	(* Init. NC parameter *)
		i:=1;
		(* Beckhoff *)
		IF sDeviceName = 'Beckhoff' THEN
			(*copy parameter value *)
			WHILE T_Axis.T_ParamFileObj[i].udiIdxGroup <> 0 DO
				CASE (T_Axis.T_ParamFileObj[i].udiIdxGroup - T_Axis.T_Config_Gen.udiNC_TaskIdxGrp) OF
				16#4000:	CASE T_Axis.T_ParamFileObj[i].udiIndexOffset OF
						(* Calibration velocity forward *)
						16#6:	T_Axis.T_Config_ObjFileValue.lrCalVelocityForward:=T_Axis.T_ParamFileObj[i].lrReal;
						(* Calibration velocity backward *)
						16#7:	T_Axis.T_Config_ObjFileValue.lrCalVelocityBackward:=T_Axis.T_ParamFileObj[i].lrReal;
						(* Maximum velocity *)
						16#27:	T_Axis.T_Config_ObjFileValue.lrMaxVelocity:=T_Axis.T_ParamFileObj[i].lrReal;
						(* Acceleration *)
						16#101:	T_Axis.T_Config_ObjFileValue.lrAcceleration:=T_Axis.T_ParamFileObj[i].lrReal;
						(* Decceleration *)
						16#102:	T_Axis.T_Config_ObjFileValue.lrDecceleration:=T_Axis.T_ParamFileObj[i].lrReal;
						(* Jerk *)
						16#103:	T_Axis.T_Config_ObjFileValue.lrJerk:=T_Axis.T_ParamFileObj[i].lrReal;
						END_CASE
				16#5000:	CASE T_Axis.T_ParamFileObj[i].udiIndexOffset OF
						(* Encoder scaling factor *)
						16#6:	T_Axis.T_Config_ObjFileValue.lrScaleFactor:=T_Axis.T_ParamFileObj[i].lrReal;
						(* SW limit negativ On/Off *)
						16#B:	T_Axis.T_Config_ObjFileValue.xSWLimitNeg:=REAL_TO_BOOL(T_Axis.T_ParamFileObj[i].lrReal);
						(* SW limit positiv On/Off *)
						16#C:	T_Axis.T_Config_ObjFileValue.xSWLimitPos:=REAL_TO_BOOL(T_Axis.T_ParamFileObj[i].lrReal);
						(* SW limit negativ value *)
						16#D:	T_Axis.T_Config_ObjFileValue.lrSWLimitNeg:=T_Axis.T_ParamFileObj[i].lrReal;
						(* SW limit position value *)
						16#E:	T_Axis.T_Config_ObjFileValue.lrSWLimitPos:=T_Axis.T_ParamFileObj[i].lrReal;
						END_CASE
				16#6000:;
				16#7000:;
				END_CASE
				(* next parameter *)
				i:=i+1;
			END_WHILE
		END_IF

		(* Maxon *)
		IF sDeviceName = 'Maxon' THEN
			(*copy parameter value *)
			WHILE T_Axis.T_ParamFileObj[i].udiIdxGroup <> 0 DO
				CASE T_Axis.T_ParamFileObj[i].udiIdxGroup  OF
				16#6083:	CASE T_Axis.T_ParamFileObj[i].udiIndexOffset OF
						(* Acceleration *)
						16#0:	T_Axis.T_Config_ObjFileValue.lrAcceleration:=T_Axis.T_ParamFileObj[i].lrReal;
						END_CASE
				16#6084:	CASE T_Axis.T_ParamFileObj[i].udiIndexOffset OF
						(* Decceleration *)
						16#0:	T_Axis.T_Config_ObjFileValue.lrDecceleration:=T_Axis.T_ParamFileObj[i].lrReal;
						END_CASE
				END_CASE
				(* next parameter *)
				i:=i+1;
			END_WHILE
		END_IF
		(* set flag done *)
		xBusy:=FALSE;
		xDone:=TRUE;
	END_IF;
END_FUNCTION_BLOCK

(* POU FB_HARDWARE/FBHW_AXIS_LIVEVALUES_BECKHOFF, ST *)
FUNCTION_BLOCK FBHW_AXIS_LIVEVALUES_BECKHOFF
VAR_INPUT
	uiActualTorque: UINT;
	arxDigitalInput: ARRAY[1..8] OF BOOL;
END_VAR
VAR_OUTPUT
END_VAR
VAR_IN_OUT
	T_Axis:ST_AXIS;
	T_AxisRefIn:NCTOPLC_AXLESTRUCT;
END_VAR
VAR
	i:INT;
END_VAR
(****************************************************************************************************************************************************)
(***********                                    This Functionblock read the actual value from the Beckhoff drive                                               ************)
(****************************************************************************************************************************************************)
(* return actual axis state *)
T_Axis.T_LiveValue.dwState:=T_AxisRefIn.nStateDWord;
(* return actual torque value *)
T_Axis.T_LiveValue.uiActualTorque:=uiActualTorque;
IF T_Axis.T_LiveValue.uiActualTorque > 16#7FFF THEN
	(* negativ value *)
	T_Axis.T_LiveValue.diActualTorqueCalc:=UINT_TO_DINT(T_Axis.T_LiveValue.uiActualTorque) - 65535;
ELSE
	(* positiv value *)
	T_Axis.T_LiveValue.diActualTorqueCalc:=UINT_TO_DINT(T_Axis.T_LiveValue.uiActualTorque);
END_IF
(* return actual velocity *)
T_Axis.T_LiveValue.lrActualVelocity:=T_AxisRefIn.fVeloIst;
(* ??? modif 06092005 *)
(* return actual position *)
IF T_Axis.T_Config_Gen.iTyp <>1 THEN
(* modulo position for rotativ axis*)
	T_Axis.T_LiveValue.lrActualPosition:=T_AxisRefIn.fModuloPosIst;
	T_Axis.T_LiveValue.lrActualPositionNotModulo:=T_AxisRefIn.fPosIst;
ELSE
(* counter value *)
	T_Axis.T_LiveValue.lrActualPosition:=T_AxisRefIn.fPosIst;
END_IF
T_Axis.T_LiveValue.lrSollPosition:=T_AxisRefIn.fPosSoll;
(* return actual position *)
(*T_Axis.T_LiveValue.lrActualPosition:=T_AxisRefIn.fPosIst;*)
(* ??? modif 06092005 *)
(* return the actual digital input state *)
T_Axis.T_LiveValue.bDigitalInput:=0;
FOR i := 0 TO 7 DO
	IF arxDigitalInput[i+1] THEN
		T_Axis.T_LiveValue.bDigitalInput:=T_Axis.T_LiveValue.bDigitalInput + MUX(i,1,2,4,8,16,32,64,128);
	END_IF
END_FOR;
END_FUNCTION_BLOCK

(* POU FB_HARDWARE/FBHW_AXIS_MULTI_BECKHOFF, ST *)
FUNCTION_BLOCK FBHW_AXIS_MULTI_BECKHOFF
VAR_INPUT
END_VAR
VAR_OUTPUT
END_VAR
VAR_IN_OUT
	T_AxisMaster:ST_AXIS;
	T_AxisSlave:ST_AXIS;
	T_AxisMasterRefIn:NCTOPLC_AXLESTRUCT;
	T_AxisSlaveRefIn:NCTOPLC_AXLESTRUCT;
END_VAR
VAR
(* block function *)
	fbAxisMasterSlaveOn:MC_GearIn;
	fbAxisMasterSlaveOff:MC_GearOut;
(* variable *)
	xGearIn:BOOL:=FALSE;
	xGearOut:BOOL:=FALSE;
	xConfirmResetFB:BOOL:=FALSE;
(* trigger *)
	RisingEdgeResetFB:R_TRIG;
	RisingEdgeExecute:R_TRIG;
END_VAR
(****************************************************************************************************************************************************)
(***********                                   This Functionblock is the driver for the Beckhoff Axis for Master/Slave                                      ************)
(****************************************************************************************************************************************************)
(* Reset block function *)
	RisingEdgeResetFB(CLK:=T_AxisMaster.T_CtrleMulti.xReset);
	IF RisingEdgeResetFB.Q THEN
	(* Init. block function *)
		fbAxisMasterSlaveOn(	Execute:=FALSE,
							Master:=T_AxisMasterRefIn,
							Slave:=T_AxisSlaveRefIn);
		fbAxisMasterSlaveOff(	Execute:=FALSE,
							Slave:=T_AxisSlaveRefIn);
	(* Init. variable *)
		xGearIn:=FALSE;
		xGearOut:=FALSE;
	(* init. structure *)
		T_AxisMaster.T_CtrleMulti.iFunction:=0;
		T_AxisMaster.T_CtrleMulti.iNumerator:=1;
		T_AxisMaster.T_CtrleMulti.uiDenominator:=1;
		T_AxisMaster.T_CtrleMulti.xDone:=FALSE;
		T_AxisMaster.T_CtrleMulti.xErr:=FALSE;
		T_AxisMaster.T_CtrleMulti.udiErrorID:=0;
		(* set done flag *)
		xConfirmResetFB:=TRUE;
		(* exit function bloc *)
		RETURN;
	ELSE
		IF xConfirmResetFB THEN
		(* confirm reset FB *)
			T_AxisMaster.T_CtrleMulti.xDone:=TRUE;
			T_AxisMaster.T_CtrleMulti.xErr:=FALSE;
			T_AxisMaster.T_CtrleMulti.udiErrorID:=0;
			(* reset variable *)
			xConfirmResetFB:=FALSE;
		END_IF
	END_IF

(* Execute *)
	RisingEdgeExecute(CLK:=T_AxisMaster.T_CtrleMulti.xExecute);
	IF RisingEdgeExecute.Q THEN
		CASE T_AxisMaster.T_CtrleMulti.iFunction OF
		(* activ master-slave *)
		1:	xGearIn:=TRUE;
		(* desactiv master-slave *)
		2: 	xGearOut:=TRUE;
		ELSE
		(* function not implemented *)
			T_AxisMaster.T_CtrleMulti.xDone:=FALSE;
			T_AxisMaster.T_CtrleMulti.xErr:=TRUE;
			T_AxisMaster.T_CtrleMulti.udiErrorID:=16#F000;
			(* exit FB *)
			RETURN;
		END_CASE
		(* Init. variable *)
		T_AxisMaster.T_CtrleMulti.xDone:=FALSE;
		T_AxisMaster.T_CtrleMulti.xErr:=FALSE;
		T_AxisMaster.T_CtrleMulti.udiErrorID:=0;
	END_IF

(* GearIn *)
	IF xGearIn THEN
		fbAxisMasterSlaveOn(	Execute:=TRUE,
							RatioNumerator:=T_AxisMaster.T_CtrleMulti.iNumerator,
							RatioDenominator:=T_AxisMaster.T_CtrleMulti.uiDenominator,
							Acceleration:=T_AxisMaster.T_CtrleSingle.lrAcceleration,
							Deceleration:=T_AxisMaster.T_CtrleSingle.lrDecceleration,
							Jerk:=T_AxisMaster.T_CtrleSingle.lrJerk,
							Master:=T_AxisMasterRefIn,
							Slave:=T_AxisSlaveRefIn);
		IF fbAxisMasterSlaveOn.InGear OR fbAxisMasterSlaveOn.Error THEN
			T_AxisMaster.T_CtrleMulti.xDone:= fbAxisMasterSlaveOn.InGear;
			T_AxisMaster.T_CtrleMulti.xErr:=fbAxisMasterSlaveOn.Error;
			T_AxisMaster.T_CtrleMulti.udiErrorID:=fbAxisMasterSlaveOn.ErrorID;
			(* set flag gearin off *)
			xGearIn:=FALSE;
		END_IF
	ELSE
		fbAxisMasterSlaveOn(	Execute:=FALSE,
							Master:=T_AxisMasterRefIn,
							Slave:=T_AxisSlaveRefIn);
	END_IF

(* GearOut *)
	IF xGearOut THEN
		fbAxisMasterSlaveOff(	Execute:=TRUE,
							Slave:=T_AxisSlaveRefIn);
		IF fbAxisMasterSlaveOff.Done OR fbAxisMasterSlaveOff.Error THEN
			T_AxisMaster.T_CtrleMulti.xDone:= fbAxisMasterSlaveOff.Done;
			T_AxisMaster.T_CtrleMulti.xErr:=fbAxisMasterSlaveOff.Error;
			T_AxisMaster.T_CtrleMulti.udiErrorID:=fbAxisMasterSlaveOff.ErrorID;
			(* set flag gearout off *)
			xGearOut:=FALSE;
		END_IF
	ELSE
		fbAxisMasterSlaveOff(	Execute:=FALSE,
							Slave:=T_AxisSlaveRefIn);
	END_IF
END_FUNCTION_BLOCK

(* POU FB_HARDWARE/FBHW_CYL_ANALOGCYLINDER, ST *)
FUNCTION_BLOCK FBHW_CYL_ANALOGCYLINDER
VAR_INPUT
	xCtrlePosOn:BOOL;
	xCtrlePosOff:BOOL;
	iAnalogIn:INT;
END_VAR
VAR_OUTPUT
	xCylinder:BOOL;
	iAnalogOut:INT;
END_VAR
VAR_IN_OUT
	T_Cylinder:ST_CYLINDER;
END_VAR
VAR
(* variable *)
	xConfirmResetFB: BOOL;
	xActivCtrle:BOOL;
	iStep:INT;
(* timer *)
	TimerOn:TON;
	TimerOff:TON;
	TimerPreOn:TON;
	TimerPreOff:TON;
	TimerOut:TON;
	TimerActiv: TON;
(* trigger *)
	RisingEdgeExecute:R_TRIG;
	RisingEdgeReset:R_TRIG;
	RisingEdgeActiv:R_TRIG;
	FallingEdgeActiv:F_TRIG;
	xFct3Activ: BOOL;
	xTmpFct3Activ: BOOL;
END_VAR
(****************************************************************************************************************************************************)
(***********                                       This Functionblock is the driver for the ToolTension Cylinder                                                    ************)
(****************************************************************************************************************************************************)
(* if function bloc set activ then Analog state will be transfered *)
	RisingEdgeActiv(CLK:=T_Cylinder.T_CtrleCyl.xFBActiv);
	FallingEdgeActiv(CLK:=T_Cylinder.T_CtrleCyl.xFBActiv);
	IF RisingEdgeActiv.Q OR FallingEdgeActiv.Q THEN
		iAnalogOut:=0;
		xCylinder:=NOT(T_Cylinder.T_Config.xActivState);
		T_Cylinder.T_CtrleCyl.T_AnalogCylinder.xActiv:= FALSE;
	END_IF
	(* transfer sensor state only if fb is activ *)
	IF T_Cylinder.T_CtrleCyl.xFBActiv THEN
		T_Cylinder.T_CtrleCyl.xStatePosOn:=xCtrlePosOn;
		T_Cylinder.T_CtrleCyl.xStatePosOff:=xCtrlePosOff;
	(* copy state value *)
		T_Cylinder.T_CtrleCyl.T_AnalogCylinder.iAnalogOut:=iAnalogOut;
	ELSE
	(* exit fb *)
		RETURN;
	END_IF

(* wait for reseting *)
	RisingEdgeReset(CLK:=T_Cylinder.T_CtrleCyl.xReset);
	IF RisingEdgeReset.Q THEN
		(* Init. timer *)
		TimerOn(IN:=TRUE,PT:=T#1ms);
		TimerOff(IN:=TRUE,PT:=T#1ms);
		TimerOut(IN:=TRUE,PT:=T#1ms);
		TimerPreOn(IN:=TRUE,PT:=T#1ms);
		TimerPreOff(IN:=TRUE,PT:=T#1ms);
		TimerActiv(IN:=TRUE,PT:=T#1ms);
	(* Init. variable *)
		xActivCtrle:=FALSE;
		iStep:=0;
		xFct3Activ:=FALSE;
		xTmpFct3Activ:=FALSE;
		T_Cylinder.T_CtrleCyl.T_AnalogCylinder.tDelayActiv:=T#0s;
		T_Cylinder.T_Config.tDelayPreOn:=T#0s;
		T_Cylinder.T_Config.tDelayPreOff:=T#0s;
	(* Init. structure *)
		T_Cylinder.T_CtrleCyl.iFunction:=0;
		T_Cylinder.T_CtrleCyl.T_AnalogCylinder.xActiv:= FALSE;
		xCylinder:=NOT(T_Cylinder.T_Config.xActivState);
		iAnalogOut:=0;
		T_Cylinder.T_CtrleCyl.xDone:=FALSE;
		T_Cylinder.T_CtrleCyl.xErr:=FALSE;
		T_Cylinder.T_CtrleCyl.udiErrorID:=16#0;
	(* confirm reset *)
		xConfirmResetFB:=TRUE;
	(* exit function *)
		RETURN;
	ELSE
		IF xConfirmResetFB THEN
		(* confirm reset FB *)
			T_Cylinder.T_CtrleCyl.xDone:=TRUE;
			T_Cylinder.T_CtrleCyl.xErr:=FALSE;
			T_Cylinder.T_CtrleCyl.udiErrorID:=16#0;
			(* init. variable *)
			xConfirmResetFB:=FALSE;
		END_IF
	END_IF

(* wait for execute *)
	RisingEdgeExecute(CLK:=T_Cylinder.T_CtrleCyl.xExecute);
	IF RisingEdgeExecute.Q THEN
		IF NOT(T_Cylinder.T_CtrleCyl.xDone) AND NOT(T_Cylinder.T_CtrleCyl.xErr) THEN
		(* can execute function if both signal are disable *)
			RETURN;
		END_IF
		CASE T_Cylinder.T_CtrleCyl.iFunction OF
		(* disable *)
		1:	iStep:=11;
		(* Activ without sensor position ctrle *)
		2:	iStep:=1;
		(* set value Analog Out = Analog In *)
		4:	iStep:=21;
		(* inverse cylinder state *)
		51:	iStep:=51;
		ELSE
			(* function not implemented *)
			iStep:=0;
			T_Cylinder.T_CtrleCyl.xDone:=FALSE;
			T_Cylinder.T_CtrleCyl.xErr:=TRUE;
			T_Cylinder.T_CtrleCyl.udiErrorID:=16#F000;
			(* exit FB *)
			RETURN;
		END_CASE
		(* Init. variable *)
		T_Cylinder.T_CtrleCyl.xDone:=FALSE;
		T_Cylinder.T_CtrleCyl.xErr:=FALSE;
		T_Cylinder.T_CtrleCyl.udiErrorID:=16#0;
		(* exit FB *)
		RETURN;
	END_IF

(* Timer activ *)
	TimerOn(IN:=TRUE,PT:=T_Cylinder.T_Config.tDelayOn);
	TimerOff(IN:=TRUE,PT:=T_Cylinder.T_Config.tDelayOff);
	TimerPreOn(IN:=TRUE,PT:=T_Cylinder.T_Config.tDelayPreOn);
	TimerPreOff(IN:=TRUE,PT:=T_Cylinder.T_Config.tDelayPreOff);
	TimerOut(IN:=TRUE,PT:=T_Cylinder.T_Config.tTimeOut);
	TimerActiv(IN:=TRUE,PT:=T_Cylinder.T_CtrleCyl.T_AnalogCylinder.tDelayActiv);
(* waiting for activ *)
	CASE iStep OF
	(* Set Analog output *)
	1:	IF (T_Cylinder.T_Config.tDelayPreOn = T#0s) THEN
			TimerOn(IN:=FALSE);
			iAnalogOut:=iAnalogIn;
			xCylinder:=T_Cylinder.T_Config.xActivState;
			T_Cylinder.T_CtrleCyl.T_AnalogCylinder.xActiv:= TRUE;
			iStep:=2;
		ELSE
			TimerPreOn(IN:=FALSE);
			iStep:=4;
		END_IF;
	(* wait for timer On *)
	2:	IF TimerOn.Q THEN
			iStep:=3;
			TimerOut(IN:=FALSE);
		END_IF
	(* control position activ *)
	3:	IF T_Cylinder.T_Config.xCtrlePosOn THEN
		(* position ctrle activ *)
			IF TimerOut.Q THEN
			(* timerout done, activ error cylinder has not activ position reached *)
				iStep:=999;
			ELSE
				IF xCtrlePosOn THEN
				(* Activ position reached, activ confirmation *)
					iStep:=90;
				END_IF
			END_IF
		ELSE
		(* no position ctrle, activ confirm *)
			iStep:=90;
		END_IF
	(* wait for timer Pre On *)
	4:	IF TimerPreOn.Q THEN
			T_Cylinder.T_Config.tDelayPreOn:=T#0s;
			iStep:=1;
		END_IF
	(* process timer Off *)
	11:	IF (T_Cylinder.T_Config.tDelayPreOff = T#0s) THEN
			TimerOff(IN:=FALSE);
			iAnalogOut:=0;
			xCylinder:=NOT(T_Cylinder.T_Config.xActivState);
			T_Cylinder.T_CtrleCyl.T_AnalogCylinder.xActiv:= FALSE;
			iStep:=12;
		ELSE
			TimerPreOff(IN:=FALSE);
			iStep:=14;
		END_IF;
	(* wait for timer Off *)
	12:	IF TimerOff.Q THEN
			iStep:=13;
			TimerOut(IN:=FALSE);
		END_IF
	(* control position inactiv *)
	13:	IF T_Cylinder.T_Config.xCtrlePosOff THEN
		(* control position activ *)
			IF TimerOut.Q THEN
			(* timerout done, activ error 'cylinder has not inactiv position reached' *)
				iStep:=998;
			ELSE
				IF xCtrlePosOff THEN
				(* inactiv position reached, activ confirmation *)
					iStep:=99;
				END_IF
			END_IF
		ELSE
		(* no control position activ, activ confirmation *)
			iStep:=99;
		END_IF
	(* wait for timer Pre Off *)
	14:	IF TimerPreOff.Q THEN
			T_Cylinder.T_Config.tDelayPreOff:=T#0s;
			iStep:=11;
		END_IF
	(* set value Analog Out = Analog In *)
	21:	xCylinder:=T_Cylinder.T_Config.xActivState;
		T_Cylinder.T_CtrleCyl.T_AnalogCylinder.xActiv:= TRUE;
		iAnalogOut:=iAnalogIn;
		iStep:=99;
	(* inverse cylinder state *)
	51:	IF T_Cylinder.T_CtrleCyl.T_AnalogCylinder.xActiv THEN
			iAnalogOut:=0;
		ELSE
			iAnalogOut:=iAnalogIn;
		END_IF;
		xCylinder:=NOT(xCylinder);
		T_Cylinder.T_CtrleCyl.T_AnalogCylinder.xActiv:=NOT(T_Cylinder.T_CtrleCyl.T_AnalogCylinder.xActiv);
		iStep:=99;
	(* test if delay activ *)
	90:	IF T_Cylinder.T_CtrleCyl.T_AnalogCylinder.tDelayActiv <> T#0s THEN
			TimerActiv(IN:=FALSE);
			iStep:=91;
		ELSE
			iStep:=99;
		END_IF
	(* wait for time delay activ *)
	91:	IF TimerActiv.Q THEN
			T_Cylinder.T_CtrleCyl.T_AnalogCylinder.tDelayActiv:=T#0s;
			iStep:=11;	(* Zylinder wird wieder deaktiviert *)
		END_IF;
	(* no ctrle position *)
	99:	T_Cylinder.T_CtrleCyl.xDone:=TRUE;
		T_Cylinder.T_CtrleCyl.xErr:=FALSE;
		T_Cylinder.T_CtrleCyl.udiErrorID:=16#0;
	(* error, cylinder not in inactiv position *)
	998:	T_Cylinder.T_CtrleCyl.xDone:=FALSE;
		T_Cylinder.T_CtrleCyl.xErr:=TRUE;
		T_Cylinder.T_CtrleCyl.udiErrorID:=16#F202;
	(* error, cylinder not in activ position *)
	999:	T_Cylinder.T_CtrleCyl.xDone:=FALSE;
		T_Cylinder.T_CtrleCyl.xErr:=TRUE;
		T_Cylinder.T_CtrleCyl.udiErrorID:=16#F201;
	END_CASE
END_FUNCTION_BLOCK

(* POU GENERAL/FB_CALC_TOOLTENSION_FORCE_NEW, ST *)
FUNCTION_BLOCK FB_CALC_TOOLTENSION_FORCE_NEW
VAR_INPUT
	rForcePistonIn:REAL;	(* in Newton *)
	rPistonDiameterD1:REAL;	(* in mm *)
	rPistonDiameterD2:REAL;	(* in mm *)
	rMaxAirpressure:REAL;		(* in bar *)
	rFactorForce:REAL;
END_VAR
VAR_OUTPUT
	iAnalogOutput:INT;		(* range 0 - 32767 *)
	rSetMaxForce:REAL;		(* in Newton *)
	rForcePistonOut:REAL;	(* in Newton *)
END_VAR
VAR
	rMaxForce: REAL;
	rAreaOutside: REAL;
	rAreaInside: REAL;
	rArea: REAL;
	rTmpMaxAirpressure: REAL;
	rTmpAnalogOut:REAL;
END_VAR
(****************************************************************************************************************************************************)
(*****       This Functionblock calculate the effective value for the servo ventil for the ToolTension which the settled force         *****)
(****************************************************************************************************************************************************)
	rAreaOutside:=((rPistonDiameterD1/2)*(rPistonDiameterD1/2))*PI;
	rAreaInside:=((rPistonDiameterD2/2)*(rPistonDiameterD2/2))*PI;
	rArea:=ABS(rAreaOutside - rAreaInside);
	rArea:=rArea / 1000000.0;	(* Umwandeln von mm^2 in m^2 *)
	rTmpMaxAirpressure:=rMaxAirpressure * 100000.0;	(* convert from bar to pascal *)
	rMaxForce:=rArea * rTmpMaxAirpressure * rFactorForce;
	rSetMaxForce:=rMaxForce;

	IF(rMaxForce = 0) THEN rMaxForce:=0.01; END_IF;	(* check divide by zero *)
	IF(rMaxForce <> 0.0) THEN
		rTmpAnalogOut:=(rForcePistonIn/rMaxForce)*32767;	(* 32767 = 10V *)
		IF (rTmpAnalogOut > 32767) THEN
			iAnalogOutput:=32767;
		ELSE
			iAnalogOutput:=REAL_TO_INT(rTmpAnalogOut);
		END_IF;
		rForcePistonOut:=rForcePistonIn;
	ELSE
		iAnalogOutput:=0;
		rForcePistonOut:=0;
	END_IF;
END_FUNCTION_BLOCK

(* POU FB_HARDWARE/FBHW_CYL_STANDARD, ST *)
FUNCTION_BLOCK FBHW_CYL_STANDARD
VAR_INPUT
	xCtrlePosOn:BOOL;
	xCtrlePosOff:BOOL;
END_VAR
VAR_OUTPUT
	xCylinder:BOOL;
END_VAR
VAR_IN_OUT
	T_Cylinder:ST_CYLINDER;
END_VAR
VAR
(* variable *)
	xConfirmResetFB:BOOL:=FALSE;
	iStep:INT;
(* timer *)
	TimerOn:TON;
	TimerOff:TON;
	TimerPreOn:TON;
	TimerPreOff:TON;
	TimerOut:TON;
	TimerActiv: TON;
(* trigger *)
	RisingEdgeActiv:R_TRIG;
	FallingEdgeActiv:F_TRIG;
	RisingEdgeReset:R_TRIG;
	RisingEdgeExecute:R_TRIG;
	TimerAfterSensor: TON;
END_VAR
(* if function bloc set activ then Analog state will be transfered *)
	RisingEdgeActiv(CLK:=T_Cylinder.T_CtrleCyl.xFBActiv);
	FallingEdgeActiv(CLK:=T_Cylinder.T_CtrleCyl.xFBActiv);
	IF RisingEdgeActiv.Q OR FallingEdgeActiv.Q THEN
	(* set Analog Out = In on the rising edge from the activ signal *)
		xCylinder:=NOT(T_Cylinder.T_Config.xActivState);
		T_Cylinder.T_CtrleCyl.T_Standard.xActivOn:= FALSE;
	END_IF

(* if bloc disable if activ signal is inactiv *)
	IF T_Cylinder.T_CtrleCyl.xFBActiv THEN
	(* copy control position state *)
		T_Cylinder.T_CtrleCyl.xStatePosOn:=xCtrlePosOn;
		T_Cylinder.T_CtrleCyl.xStatePosOff:=xCtrlePosOff;
	ELSE
	(* exit FB *)
		T_Cylinder.T_CtrleCyl.xStatePosOn:=xCtrlePosOn;
		T_Cylinder.T_CtrleCyl.xStatePosOff:=xCtrlePosOff;
		RETURN;
	END_IF

(* wait for reseting *)
	RisingEdgeReset(CLK:=T_Cylinder.T_CtrleCyl.xReset);
	IF RisingEdgeReset.Q THEN
		(* Init. timer *)
		TimerOn(IN:=TRUE,PT:=T#1ms);
		TimerOff(IN:=TRUE,PT:=T#1ms);
		TimerPreOn(IN:=TRUE,PT:=T#1ms);
		TimerPreOff(IN:=TRUE,PT:=T#1ms);
		TimerOut(IN:=TRUE,PT:=T#1ms);
	(* Init. variable *)
		iStep:=0;
	(* Init. structure *)
		T_Cylinder.T_CtrleCyl.iFunction:=0;
		T_Cylinder.T_CtrleCyl.T_Standard.xActivOn:=FALSE;
		xCylinder:=NOT(T_Cylinder.T_Config.xActivState);
		T_Cylinder.T_CtrleCyl.xDone:=FALSE;
		T_Cylinder.T_CtrleCyl.xErr:=FALSE;
		T_Cylinder.T_CtrleCyl.udiErrorID:=16#0;
	(* confirm reset *)
		xConfirmResetFB:=TRUE;
	(* exit function *)
		RETURN;
	ELSE
		IF xConfirmResetFB THEN
		(* confirm reset FB *)
			T_Cylinder.T_CtrleCyl.xDone:=TRUE;
			T_Cylinder.T_CtrleCyl.xErr:=FALSE;
			T_Cylinder.T_CtrleCyl.udiErrorID:=16#0;
			(* reset variable *)
			xConfirmResetFB:=FALSE;
		END_IF
	END_IF

(* if bloc disable if activ signal is inactiv *)
	IF NOT(T_Cylinder.T_CtrleCyl.xFBActiv) THEN
		RETURN;
	END_IF

(* wait for execute *)
	RisingEdgeExecute(CLK:=T_Cylinder.T_CtrleCyl.xExecute);
	IF RisingEdgeExecute.Q THEN
		IF NOT(T_Cylinder.T_CtrleCyl.xDone) AND NOT(T_Cylinder.T_CtrleCyl.xErr) THEN
		(* can execute function if both signal are disable *)
			RETURN;
		END_IF
		CASE T_Cylinder.T_CtrleCyl.iFunction OF
		(* disable *)
		1:	iStep:=11;
		(* Activ without sensor position ctrle *)
		2:	iStep:=1;
		(* inverse cylinder state *)
		51:	iStep:=51;
		ELSE
			(* function not implemented *)
			iStep:=0;
			T_Cylinder.T_CtrleCyl.xDone:=FALSE;
			T_Cylinder.T_CtrleCyl.xErr:=TRUE;
			T_Cylinder.T_CtrleCyl.udiErrorID:=16#F000;
			(* exit FB *)
			RETURN;
		END_CASE
		(* Init. variable *)
		T_Cylinder.T_CtrleCyl.xDone:=FALSE;
		T_Cylinder.T_CtrleCyl.xErr:=FALSE;
		T_Cylinder.T_CtrleCyl.udiErrorID:=16#0;
		(* exit FB *)
		RETURN;
	END_IF

(* Timer activ *)
	TimerOn(IN:=TRUE,PT:=T_Cylinder.T_Config.tDelayOn);
	TimerOff(IN:=TRUE,PT:=T_Cylinder.T_Config.tDelayOff);
	TimerPreOn(IN:=TRUE,PT:=T_Cylinder.T_Config.tDelayPreOn);
	TimerPreOff(IN:=TRUE,PT:=T_Cylinder.T_Config.tDelayPreOff);
	TimerOut(IN:=TRUE,PT:=T_Cylinder.T_Config.tTimeOut);
	TimerActiv(IN:=TRUE,PT:=T_Cylinder.T_CtrleCyl.T_Standard.tDelayActiv);
	TimerAfterSensor(IN:=TRUE,PT:=T_Cylinder.T_CtrleCyl.T_Standard.tDelayAfterSensor);
(* waiting for activ *)
	CASE iStep OF
	(* process timer On *)
	1:	IF (T_Cylinder.T_Config.tDelayPreOn = T#0s) THEN
			TimerOn(IN:=FALSE);
			xCylinder:=T_Cylinder.T_Config.xActivState;
			T_Cylinder.T_CtrleCyl.T_Standard.xActivOn:=TRUE;
			iStep:=2;
		ELSE
			TimerPreOn(IN:=FALSE);
			iStep:=4;
		END_IF;
	(* wait for timer On *)
	2:	IF TimerOn.Q THEN
			iStep:=3;
			TimerOut(IN:=FALSE);
		END_IF
	(* control position activ *)
	3:	IF T_Cylinder.T_Config.xCtrlePosOn THEN
		(* position ctrle activ *)
			IF TimerOut.Q THEN
			(* timerout done, activ error cylinder has not activ position reached *)
				iStep:=999;
			ELSE
				IF xCtrlePosOn THEN
				(* Activ position reached, activ confirmation *)
					iStep:=80;
				END_IF
			END_IF
		ELSE
		(* no position ctrle, activ confirm *)
			iStep:=90;
		END_IF
	(* wait for timer Pre On *)
	4:	IF TimerPreOn.Q THEN
			T_Cylinder.T_Config.tDelayPreOn:=T#0s;
			iStep:=1;
		END_IF
	(* process timer Off *)
	11:	IF (T_Cylinder.T_Config.tDelayPreOff = T#0s) THEN
			TimerOff(IN:=FALSE);
			xCylinder:=NOT(T_Cylinder.T_Config.xActivState);
			T_Cylinder.T_CtrleCyl.T_Standard.xActivOn:=FALSE;
			iStep:=12;
		ELSE
			TimerPreOff(IN:=FALSE);
			iStep:=14;
		END_IF;
	(* wait for timer Off *)
	12:	IF TimerOff.Q THEN
			iStep:=13;
			TimerOut(IN:=FALSE);
		END_IF
	(* control position inactiv *)
	13:	IF T_Cylinder.T_Config.xCtrlePosOff THEN
		(* control position activ *)
			IF TimerOut.Q THEN
			(* timerout done, activ error 'cylinder has not inactiv position reached' *)
				iStep:=998;
			ELSE
				IF xCtrlePosOff THEN
				(* inactiv position reached, activ confirmation *)
					iStep:=85;
				END_IF
			END_IF
		ELSE
		(* no control position activ, activ confirmation *)
			iStep:=99;
		END_IF
	(* wait for timer Pre Off *)
	14:	IF TimerPreOff.Q THEN
			T_Cylinder.T_Config.tDelayPreOff:=T#0s;
			iStep:=11;
		END_IF
	(* inverse cylinder state *)
	51:	xCylinder:=NOT(xCylinder);
		T_Cylinder.T_CtrleCyl.T_Standard.xActivOn:=NOT(T_Cylinder.T_CtrleCyl.T_Standard.xActivOn);
		iStep:=99;
	80:	IF (T_Cylinder.T_CtrleCyl.T_Standard.tDelayAfterSensor <> T#0s) THEN
			TimerAfterSensor(IN:=FALSE);
			iStep:=81;
		ELSE
			iStep:=90;
		END_IF;
	(* wait for time after sensor *)
	81:	IF TimerAfterSensor.Q THEN
			iStep:=90;
		END_IF
	85:	IF (T_Cylinder.T_CtrleCyl.T_Standard.tDelayAfterSensor <> T#0s) THEN
			TimerAfterSensor(IN:=FALSE);
			iStep:=86;
		ELSE
			iStep:=99;
		END_IF;
	(* wait for time after sensor *)
	86:	IF TimerAfterSensor.Q THEN
			iStep:=99;
		END_IF
	(* test if delay activ *)
	90:	IF T_Cylinder.T_CtrleCyl.T_Standard.tDelayActiv <> T#0s THEN
			TimerActiv(IN:=FALSE);
			iStep:=98;
		ELSE
			iStep:=99;
		END_IF
	(* wait for time delay activ *)
	98:	IF TimerActiv.Q THEN
		(* activ time is over, set variable off *)
			xCylinder:=NOT(T_Cylinder.T_Config.xActivState);
			T_Cylinder.T_CtrleCyl.T_Standard.xActivOn:=FALSE;
			iStep:=99;
		END_IF
	(* process end *)
	99:	T_Cylinder.T_CtrleCyl.xDone:=TRUE;
		T_Cylinder.T_CtrleCyl.xErr:=FALSE;
		T_Cylinder.T_CtrleCyl.udiErrorID:=16#0;
	(* error, cylinder not in inactiv position *)
	998:	T_Cylinder.T_CtrleCyl.xDone:=FALSE;
		T_Cylinder.T_CtrleCyl.xErr:=TRUE;
		T_Cylinder.T_CtrleCyl.udiErrorID:=16#F202;
	(* error, cylinder not in activ position *)
	999:	T_Cylinder.T_CtrleCyl.xDone:=FALSE;
		T_Cylinder.T_CtrleCyl.xErr:=TRUE;
		T_Cylinder.T_CtrleCyl.udiErrorID:=16#F201;
	END_CASE
END_FUNCTION_BLOCK

(* POU FB_HARDWARE/FBHW_AXIS_FU, ST *)
FUNCTION_BLOCK FBHW_AXIS_FU
VAR_INPUT
	IxReady:BOOL;
	IxError:BOOL;
	IxSpeedOK:BOOL;

	IiAActualSpeed:INT;
	IiAActualLoad:INT;
END_VAR
VAR_IN_OUT
	T_Axis:ST_AXIS;
END_VAR
VAR_OUTPUT
	QxEnable:BOOL;
	QxStart:BOOL;
	QxCCW:BOOL;
	QxReset:BOOL;
	QxReleaseBrake:BOOL;
	QxQuickStop:BOOL;

	QiASpeed:INT;
END_VAR
VAR
	xReset:BOOL;
	xPowerOn:BOOL;
	xPowerOff:BOOL;
	xStop:BOOL;
	xMoveVel:BOOL;
	iStep:INT;


	bCounter:BYTE:=1;
	diSpeedFilter:DINT;
	diLoadFilter:DINT;
END_VAR
(* Reset *)
IF T_Axis.T_CtrleSingle.xReset OR xReset THEN
	xPowerOn:=FALSE;
	xPowerOff:=FALSE;
	xStop:=FALSE;
	xMoveVel:=FALSE;

	QxEnable:=FALSE;
	QxQuickStop:=TRUE;

	IF IxError THEN
		QxReset:=TRUE;
	ELSE
		QxReset:=FALSE;
		xReset:=FALSE;
		T_Axis.T_CtrleSingle.xReset:=FALSE;
		T_Axis.T_CtrleSingle.xDone:=TRUE;
		T_Axis.T_CtrleSingle.xErr:=FALSE;
		T_Axis.T_CtrleSingle.udiErrorID:=0;
	END_IF
END_IF

(* Execute *)
IF T_Axis.T_CtrleSingle.xExecute THEN
	T_Axis.T_CtrleSingle.xExecute:=FALSE;
	T_Axis.T_CtrleSingle.xDone:=FALSE;
	T_Axis.T_CtrleSingle.xErr:=FALSE;
	T_Axis.T_CtrleSingle.udiErrorID:=0;


	CASE T_Axis.T_CtrleSingle.iFunction OF
	(* Reset *)
	1:	xReset:=TRUE;
	(* Power ON *)
	3:	xPowerOn:=TRUE;
	(* Power OFF *)
	4:	xPowerOff:=TRUE;
	(* Stop *)
	5:	xStop:=TRUE;
	(* Move Velocity *)
	6:	xMoveVel:=TRUE;
	END_CASE

	iStep:=1;
END_IF



(* Monitoring *)
T_Axis.T_CtrleSingle.xReady:=IxReady;
T_Axis.T_CtrleSingle.xPower:=IxReady AND QxEnable;
T_Axis.T_CtrleSingle.xNotMoving:=NOT(QxStart);

diSpeedFilter:=diSpeedFilter + IiAActualSpeed;
diLoadFilter:=diLoadFilter + IiAActualLoad;
bCounter:=bCounter + 1;
IF (bCounter >= 100)THEN
	diSpeedFilter:=diSpeedFilter / bCounter;
	diLoadFilter:=diLoadFilter / bCounter;
	bCounter:=1;

	IF T_Axis.T_CtrleSingle.xNotMoving AND NOT(xStop) THEN
		T_Axis.T_LiveValue.lrActualVelocity:=0.0;
	ELSE
		T_Axis.T_LiveValue.lrActualVelocity:=30000.0 / 32767.0 * diSpeedFilter;
	END_IF
	T_Axis.T_LiveValue.uiActualTorque:=LREAL_TO_UINT(100 / 32767.0 * diLoadFilter);
	IF (T_Axis.T_LiveValue.uiActualTorque < 0) THEN T_Axis.T_LiveValue.uiActualTorque:=0; END_IF
END_IF


(******************************************************************************************************************************************)
(* Function *)
(******************************************************************************************************************************************)
(* End Function *)
CASE iStep OF
90:	T_Axis.T_CtrleSingle.xDone:=TRUE;
	iStep:=0;
	xReset:=FALSE;
	xPowerOn:=FALSE;
	xPowerOff:=FALSE;
	xStop:=FALSE;
	xMoveVel:=FALSE;
END_CASE



(* Reset *)
(*IF xReset THEN
	CASE iStep OF
	1:	T_Axis.T_CtrleSingle.xReset:=FALSE;
		T_Axis.T_CtrleSingle.xDone:=TRUE;
		T_Axis.T_CtrleSingle.xErr:=FALSE;
		T_Axis.T_CtrleSingle.udiErrorID:=0;
		QxEnable:=FALSE;

		xReset:=FALSE;
		xPowerOn:=FALSE;
		xPowerOff:=FALSE;
		xStop:=FALSE;
		xMoveVel:=FALSE;

		iStep:=90;
	END_CASE
END_IF*)

(* Power ON *)
IF xPowerOn THEN
	CASE iStep OF
	1:	QxEnable:=IxReady;
		iStep:=90;
	END_CASE
END_IF



(* Power OFF *)
IF xPowerOff THEN
	CASE iStep OF
	1:	QxEnable:=FALSE;
		iStep:=90;
	END_CASE
END_IF



(* Stop *)
IF xStop THEN
	CASE iStep OF
	1:	QxStart:=FALSE;
		iStep:=iStep + 1;
	2:	(*IF NOT(IxSpeedOK) THEN*)
			iStep:=iStep + 1;
		(*END_IF*)
	3:	(*IF IxSpeedOK THEN*)
			iStep:=iStep + 1;
		(*END_IF*)
	4:	iStep:=90;
	END_CASE
END_IF


QiASpeed:=LREAL_TO_INT(32767.0 / 30000.0 * T_Axis.T_CtrleSingle.lrVelocity);
(* Move Velocity *)
IF xMoveVel THEN
	CASE iStep OF
	1:	QiASpeed:=LREAL_TO_INT(32767.0 / 30000.0 *T_Axis.T_CtrleSingle.lrVelocity);
		QxStart:=TRUE;
		iStep:=iStep + 1;
	2:	(*IF NOT(IxSpeedOK) THEN*)
			iStep:=iStep + 1;
		(*END_IF*)
	3:	(*IF IxSpeedOK THEN*)
			iStep:=iStep + 1;
		(*END_IF*)
	4:	iStep:=90;
	END_CASE
END_IF
END_FUNCTION_BLOCK

(* POU FB_HARDWARE/FBHW_SENSOR_TILT, ST *)
FUNCTION_BLOCK FBHW_SENSOR_TILT
VAR_INPUT
	IiATiltSensor:INT;
	rMaxV:REAL;
	r0DegV:REAL;
	rPlus90DegV:REAL;
	rMin90DegV:REAL;
END_VAR
VAR_OUTPUT
	rActualDegree:REAL;
END_VAR
VAR
	r0DegDigit:REAL;
	rPlus90DegDigit:REAL;
	rMinus90DegDigit:REAL;

	bCounter:BYTE:=1;
	diFilter:DINT;

	(* Test *)
	rActDegree:REAL;
	iTmp:INT;
END_VAR
r0DegDigit:=32767.0 / rMaxV * r0DegV;
rPlus90DegDigit:=32767.0 / rMaxV * rPlus90DegV;
rMinus90DegDigit:=32767.0 / rMaxV * rMin90DegV;


diFilter:=diFilter + IiATiltSensor;
bCounter:=bCounter + 1;
IF (bCounter >= 100)THEN
	diFilter:=diFilter / bCounter;
	bCounter:=1;

	IF (IiATiltSensor > r0DegDigit) THEN		(* + Bereich *)
		rActualDegree:=90.0 / (rPlus90DegDigit - r0DegDigit) * (diFilter(*IiATiltSensor*) - r0DegDigit);
	ELSIF (IiATiltSensor < r0DegDigit) THEN	(* - Bereich *)
		rActualDegree:=90.0 / (r0DegDigit - rMinus90DegDigit) * (r0DegDigit - diFilter(*IiATiltSensor*));
		rActualDegree:=rActualDegree * -1.0;
	ELSE
		rActualDegree:=0.0;
	END_IF
END_IF


(* Test *)
IF (iTmp > r0DegDigit) THEN		(* + Bereich *)
	rActDegree:=90.0 / (rPlus90DegDigit - r0DegDigit) * (iTmp - r0DegDigit);
ELSIF (iTmp < r0DegDigit) THEN	(* - Bereich *)
	rActDegree:=90.0 / (r0DegDigit - rMinus90DegDigit) * (r0DegDigit - iTmp);
	rActDegree:=rActDegree * -1.0;
ELSE
	rActDegree:=0.0;
END_IF
END_FUNCTION_BLOCK

(* POU PRG_TWINSAFE, FBD *)
PROGRAM PRG_TWINSAFE
VAR
	TwinSAFEinputKlemme1: TwinSAFE_input;
	TwinSAFEinputKlemme2: TwinSAFE_input;
	TwinSAFEinputKlemme3: TwinSAFE_input;
END_VAR
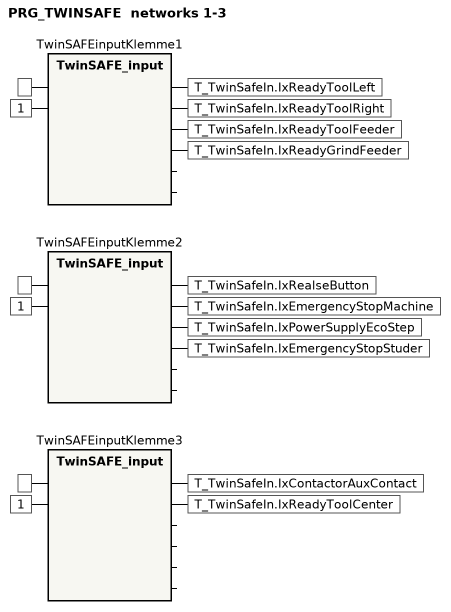
_FBD_ (* Function Block Diagram *)
NETWORK 1 (* Read of the TwinSAFE inputs *)
	TwinSAFEinputKlemme1:TwinSAFE_input(, 1, out 2 => T_TwinSafeIn.IxReadyToolRight, out 3 => T_TwinSafeIn.IxReadyToolFeeder, out 4 => T_TwinSafeIn.IxReadyGrindFeeder) => T_TwinSafeIn.IxReadyToolLeft
NETWORK 2 (* Read of the TwinSAFE inputs *)
	TwinSAFEinputKlemme2:TwinSAFE_input(, 1, out 2 => T_TwinSafeIn.IxEmergencyStopMachine, out 3 => T_TwinSafeIn.IxPowerSupplyEcoStep, out 4 => T_TwinSafeIn.IxEmergencyStopStuder) => T_TwinSafeIn.IxRealseButton
NETWORK 3 (* Read of the TwinSAFE inputs *)
	TwinSAFEinputKlemme3:TwinSAFE_input(, 1, out 2 => T_TwinSafeIn.IxReadyToolCenter) => T_TwinSafeIn.IxContactorAuxContact
_END_FBD_
END_PROGRAM

(* POU PRG_USB_IO_PANEL, ST *)
PROGRAM PRG_USB_IO_PANEL
VAR
(* Panel tastatur *)
	(* function bloc *)
	fbCtrlePanel_IO:FBHW_PANEL_IO;
	(* IO connection *)

	IarxCtrlePanelButton AT %I* : ARRAY[1..10] OF BOOL;
	QarxCtrlePanelLed AT %Q* : ARRAY[1..10] OF BOOL;
END_VAR
(****************************************************************************************************************************************************)
(***********                This Programm Unit make the connection for read and set the ControlPanel Led and Button               ************)
(****************************************************************************************************************************************************)
(* Call FB *)
	fbCtrlePanel_IO(	arxButton:=IarxCtrlePanelButton,
					T_CtrlePanel:=T_CtrlePanel,
					arxLed=>QarxCtrlePanelLed);
END_PROGRAM

(* POU FB_HARDWARE/FBHW_PANEL_IO, ST *)
FUNCTION_BLOCK FBHW_PANEL_IO
VAR_INPUT
	arxButton:ARRAY[1..10] OF BOOL;
END_VAR
VAR_OUTPUT
	arxLed:ARRAY[1..10] OF BOOL;
END_VAR
VAR_IN_OUT
	T_CtrlePanel:ST_CTRLEPANEL;
END_VAR
VAR
(* variable *)
	xConfirmResetFB:BOOL;
	xConfirmFct:BOOL;
	i: INT;
	si: SINT;
(* trigger *)
	RisingEdgeExecute:R_TRIG;
	RisingEdgeReset:R_TRIG;
END_VAR
(****************************************************************************************************************************************************)
(***********                                            This Functionblock is for manage the IO's of the ControlPanel                                             ************)
(****************************************************************************************************************************************************)
(* reset function bloc *)
	RisingEdgeReset(CLK:=T_CtrlePanel.xReset);
	IF RisingEdgeReset.Q THEN
	(* reset output *)
		FOR i := 1 TO 10 DO
			arxLed[i]:=FALSE;
		END_FOR
	(* init. structure *)
		T_CtrlePanel.iFunction:=0;
		T_CtrlePanel.xDone:=FALSE;
		T_CtrlePanel.xErr:=FALSE;
		T_CtrlePanel.udiErrorID:=0;
		T_CtrlePanel.udiButton:=0;
		T_CtrlePanel.udiLED:=0;
	(* confirm reset *)
		xConfirmResetFB:=TRUE;
	(* exit fb *)
		RETURN;
	ELSE
		IF xConfirmResetFB THEN
		(* confirm reset FB *)
			T_CtrlePanel.xDone:=TRUE;
			T_CtrlePanel.xErr:=FALSE;
			T_CtrlePanel.udiErrorID:=0;
			(* Init. variable *)
			xConfirmResetFB:=FALSE;
		END_IF
	END_IF

(* Switch on/off the Led from the control panel *)
	RisingEdgeExecute(CLK:=T_CtrlePanel.xExecute);
	IF RisingEdgeExecute.Q THEN
		CASE T_CtrlePanel.iFunction OF
		(* switch off a specific LED off *)
		-10..-1:	IF arxLed[ABS(T_CtrlePanel.iFunction)] THEN
					arxLed[ABS(T_CtrlePanel.iFunction)]:=FALSE;
					T_CtrlePanel.udiLED:=T_CtrlePanel.udiLED - MUX(ABS(T_CtrlePanel.iFunction)-1,1,2,4,8,16,32,64,128,256,512);
				END_IF
		(* switch off all the LED *)
		0:	FOR i := 1 TO 10 DO
				arxLed[i]:=FALSE;
			END_FOR
			T_CtrlePanel.udiLED:=0;
		(* switch on a specific Led on *)
		1..10:	IF NOT(arxLed[T_CtrlePanel.iFunction]) THEN
					arxLed[T_CtrlePanel.iFunction]:=TRUE;
					T_CtrlePanel.udiLED:=T_CtrlePanel.udiLED + MUX(T_CtrlePanel.iFunction-1,1,2,4,8,16,32,64,128,256,512);
				END_IF
		ELSE
			(* function not implemented *)
			T_CtrlePanel.xDone:=FALSE;
			T_CtrlePanel.xErr:=TRUE;
			T_CtrlePanel.udiErrorID:=16#F000;
			(* exit FB *)
			RETURN;
		END_CASE
		(* Init. variable *)
		T_CtrlePanel.xDone:=FALSE;
		T_CtrlePanel.xErr:=FALSE;
		T_CtrlePanel.udiErrorID:=16#0;
		(* activ confirm *)
		xConfirmFct:=TRUE;
		(* exit FB *)
		RETURN;
	END_IF

(* return the button state *)
	T_CtrlePanel.udiButton:=0;
	FOR i := 0 TO 9 DO
		IF arxButton[i+1] THEN
			T_CtrlePanel.udiButton:=T_CtrlePanel.udiButton + MUX(i,1,2,4,8,16,32,64,128,256,512);
		END_IF
	END_FOR

(* set the led state *)
	FOR si := 0 TO 9 DO
		IF GETBIT32(T_CtrlePanel.udiLED,si) <> 16#0 THEN
			arxLed[si+1]:=TRUE; ELSE arxLed[si+1]:=FALSE; END_IF
	END_FOR

(* wait to confirm *)
	IF xConfirmFct THEN
		T_CtrlePanel.xDone:=TRUE;
		T_CtrlePanel.xErr:=FALSE;
		T_CtrlePanel.udiErrorID:=16#0;
		(* reset variable *)
		xConfirmFct:=FALSE;
	END_IF
END_FUNCTION_BLOCK

(* POU GENERAL/FB_CALC_TOOLTENSION_FORCE, ST *)
FUNCTION_BLOCK FB_CALC_TOOLTENSION_FORCE
VAR_INPUT
	rForcePistonIn:REAL;	(* in Newton *)
	rPistonDiameterD:REAL;	(* in mm *)
	rMaxAirpressure:REAL;		(* in bar *)
END_VAR
VAR_OUTPUT
	iAnalogOutput:INT;		(* range 0 - 32767 *)
	rSetMaxForce:REAL;		(* in Newton *)
	rForcePistonOut:REAL;		(* in Newton *)
END_VAR
VAR
	rMaxForce: REAL;
	rAreaOutside: REAL;
	rArea: REAL;
	rTmpMaxAirpressure: REAL;
	rTmpAnalogOut:REAL;
END_VAR
(****************************************************************************************************************************************************)
(*****       This Functionblock calculate the effective value for the servo ventil for the ToolTension which the settled force         *****)
(****************************************************************************************************************************************************)
	rAreaOutside:=((rPistonDiameterD/2)*(rPistonDiameterD/2))*PI;
	rArea:=rAreaOutside;
	rArea:=rArea / 1000000.0;	(* calculate from mm^2 to m^2 *)
	rTmpMaxAirpressure:=rMaxAirpressure * 100000.0;	(* convert from bar to pascal *)
	rMaxForce:=rArea * rTmpMaxAirpressure;
	rSetMaxForce:=rMaxForce;
	IF(rMaxForce = 0) THEN rMaxForce:=0.01; END_IF;	(* check divide by zero *)
	IF(rMaxForce <> 0.0) THEN
		rTmpAnalogOut:=(rForcePistonIn/rMaxForce)*32767;	(* 32767 = 10V *)
		IF (rTmpAnalogOut > 32767) THEN
			iAnalogOutput:=32767;
		ELSE
			iAnalogOutput:=REAL_TO_INT(rTmpAnalogOut);
		END_IF;
		rForcePistonOut:=rForcePistonIn;
	ELSE
		iAnalogOutput:=0;
		rForcePistonOut:=0;
	END_IF;
END_FUNCTION_BLOCK

(* POU PRG_VISU_LAYER5/FB_VISU/rFctCalcMaxToolDiameter, ST *)
FUNCTION rFctCalcMaxToolDiameter : REAL
VAR_INPUT
	rDistanceD1:REAL;		(* distance d1 of the prisma *)
	rDistanceD2:REAL;		(* distance d2 of the prisma *)
	rAnglePrism:REAL;		(* angle of the prisma *)
END_VAR
VAR
	rTmp: REAL;
	rTmpMaxDia: REAL;
END_VAR
(****************************************************************************************************************************************************)
(***********                    This Function calculate the maximum of the tooldiameter in case of the settled prisma                      ************)
(****************************************************************************************************************************************************)
rTmp:=SIN((90 - rAnglePrism/2) * PI/180);
IF rTmp <> 0 THEN
	rTmpMaxDia:=rDistanceD1/rTmp;
ELSE
	rTmpMaxDia:=0;
END_IF;
rFctCalcMaxToolDiameter:=rTmpMaxDia;
END_FUNCTION

(* POU PRG_VISU_LAYER5/FB_VISU/rFctCalcMinToolDiameter, ST *)
FUNCTION rFctCalcMinToolDiameter : REAL
VAR_INPUT
	rDistanceD1:REAL;		(* distance d1 of the prisma *)
	rDistanceD2:REAL;		(* distance d2 of the prisma *)
	rAnglePrism:REAL;		(* angle of the prisma *)
	bStateInputPrisma:BYTE;	(* choice of selected prisma *)
END_VAR
VAR
	rTmp: REAL;
	rTmp1: REAL;
	rMinD1_1: REAL;
	rMinD1_2: REAL;
	rReturnValue: REAL;
END_VAR
(****************************************************************************************************************************************************)
(***********                    This Function calculate the minimum of the tooldiameter in case of the settled prisma                      ************)
(****************************************************************************************************************************************************)
rFctCalcMinToolDiameter:=0;
rTmp:=TAN((rAnglePrism/2)*PI/180);
rTmp1:=SIN((rAnglePrism/2)*PI/180);
IF (rTmp <> 0) AND (rTmp1 <> 0) THEN
	rMinD1_1:=rDistanceD1/(rTmp * (1 + 1/rTmp1));
END_IF;
rMinD1_2:=rDistanceD2;
IF (bStateInputPrisma = 0) OR (bStateInputPrisma = 1) THEN
	IF (rMinD1_1 >= rMinD1_2) THEN
		rReturnValue:=rMinD1_1;
	ELSE
		rReturnValue:=rMinD1_2;
	END_IF;
ELSE
	rReturnValue:=rMinD1_1;
END_IF;
rFctCalcMinToolDiameter:=rReturnValue;
END_FUNCTION

(* POU PRG_VISU_LAYER5/FB_VISU/rFctCalcPrismaFactor, ST *)
FUNCTION rFctCalcPrismaFactor : REAL
VAR_INPUT
	rAnglePrism:REAL;	(* angle of the prisma *)
END_VAR
VAR
	rFactorPrisma: REAL;
END_VAR
(****************************************************************************************************************************************************)
(***********     This Function calculate the correctur factor for the GrindFeeder Axis dependent of the settled prisma         ************)
(****************************************************************************************************************************************************)
rFctCalcPrismaFactor:=0.0;
rFactorPrisma:=(1 + SIN((rAnglePrism / 2.0) * PI/180)) / (2.0 * SIN((rAnglePrism / 2.0) * PI / 180.0));
(* Auf 5 Kommastellen runden *)
rFactorPrisma:=	STRING_TO_REAL(	LREAL_TO_FMTSTR(	in:=rFactorPrisma,
														iPrecision:=5,
														bRound:=TRUE));

rFctCalcPrismaFactor:=rFactorPrisma;
END_FUNCTION
